(* LS Electric XG5000 project: PID_project *)
(* PLC LSPLC *)
(* module base 0 slot 0: Input/Output Module:XEM-DN/DP32HP (DC 24V Input, Transistor Output, 32 Contacts) *)
(* module base 0 slot 1: Internal Positioning:XBF-PO06E (Open Collector Type, 6 Axis) *)
(* module base 0 slot 2: Input Module:XBE-DC16A/B (DC 24V Input, 16 Contacts / DC12/24V Input, 16 Contacts) *)
(* module base 0 slot 3: Output Module:XBE-RY16A (Relay Output, 16 Contacts (2A, No Varistor/Varistor)) *)
(* module base 0 slot 4: Analog Input Module:XBF-AD04C (A/D Voltage/Current Input Type, 4 Channels, 14bit) *)
(* module base 0 slot 5: Analog Output Module:XBF-DV04C (D/A Voltage Output Type, 4 Channels, 14bit) *)
VAR_GLOBAL
    _04_CH0_DATA AT %UW0.4.2 : WORD; (* Analog Input Module: CH0 Output *)
    _05_CH0_DATA AT %UW0.5.3 : WORD; (* Analog Output Module: CH0 Input *)
    _05_CH0_OUTEN AT %UX0.5.32 : BOOL; (* Analog Output Module: CH0 Output Enable *)
END_VAR

PROGRAM PID_ST (* task: Scan Program *)
(* PID program example in ST *)
VAR RETAIN
    D0_Saved_Value : REAL := 0; (* D value from auto-tune for PID0.  It is a retained variable. *)
    I0_Saved_Value : REAL := 0; (* I value from auto-tune for PID0.  It is a retained variable *)
    P0_Saved_Value : REAL := 1.0; (* P value from auto-tune for PID0.  It is a retained variable *)
    PID0_AutoTune_Completed : BOOL; (* status that auto-tune has been done for PID0.  It is a retained variable. *)
END_VAR
VAR
    Enable_PID0 : BOOL; (* command to enable PID0 *)
    INST_PID0AT : PIDAT; (* instance of auto-tune function block *)
    INST_PID0RUN : PIDRUN; (* instance of PID0 run function block *)
    INST_R_TRIG : R_TRIG;
    PID0_AutoTune_Status : WORD; (* status word of the auto-tune function *)
    PID0_Status : WORD; (* status word of PID0 *)
    Program_Step : USINT := 0; (* program step for PID0 *)
    Rising_Edge_AutoTune : BOOL; (* rising edge of auto-tune command *)
    Run_Auto_Tune : BOOL; (* command to run auto tune *)
END_VAR
VAR_EXTERNAL
    _04_CH0_DATA : WORD; (* AT %UW0.4.2 *) (* Analog Input Module: CH0 Output *)
    _05_CH0_DATA : WORD; (* AT %UW0.5.3 *) (* Analog Output Module: CH0 Input *)
    _05_CH0_OUTEN : BOOL; (* AT %UX0.5.32 *) (* Analog Output Module: CH0 Output Enable *)
END_VAR
(* 
AutomationDirect.com has provided this code for convenience. This sample code is provided "as-is" with no expressed or implied warranty. 
 If the end user includes any of the sample code (in whole or part), it is the user's responsibility to completely modify, integrate, and test any code to ensure it meets all system and 
 safety requirements for the intended application or system.
 *)

//Enable Analog Out CH0 to use it.
_05_CH0_OUTEN := TRUE;

// Clear Analog Out CH0 value if PID0 is disabled.
IF(Enable_PID0 = FALSE) THEN
	_05_CH0_DATA := 0;
END_IF;	

//Moves motor value from analog input ch0 in slot4 to auto-tuning Loop0 current value input device and PID Loop 0 current value input device.
_AT00_PV := _04_CH0_DATA;
_PID00_PV := _04_CH0_DATA;

 INST_R_TRIG(CLK:=Run_Auto_Tune, Q=>Rising_Edge_AutoTune);

CASE Program_Step OF 	
	//Program Step0:  Wait for PID0_Enable to be high.  If auto-tune has been completed, go to PID control in step 50.  If not complete, perform auto-tune in step 10.
	0:
		IF  (Rising_Edge_AutoTune = TRUE) THEN
			Program_Step := 10;
			
		ELSIF (Enable_PID0 = TRUE) AND (PID0_AutoTune_Completed = TRUE) THEN
			Program_Step := 50;
			
		END_IF;	
		
	//Program Step 10: Start Auto-Tune for PID0.  Also, moves output of auto-tuning to CH0 data of analog output module. When Complete go to Step 20.	
	10:	
		_AT00_SV := 2500;  //users set this to a value appropriate for your system
		INST_PID0AT(REQ:=TRUE, BLOCK:=0, LOOP:=0, AT_STAT=>PID0_AutoTune_Status);
		_05_CH0_DATA := _AT00_MV;
		
		IF (_AT00_STATUS = 128) THEN
			PID0_AutoTune_Completed := TRUE;
			Program_Step := 20;
		END_IF;	
	
	//Program Step 20:  Save Auto-tune values to retained variables.  return to step 0 because auto-tune is complete
	20:	
		P0_Saved_Value := _AT00_K_p;
		I0_Saved_Value := _AT00_T_i;
		D0_Saved_Value := _AT00_T_d;
		Program_Step := 0;
		
	//Program Step 50:  Copy saved auto-tune values to PID0 P,I,D values.  move to step 60 to start PID0.	
	50:
		_PID00_K_p := P0_Saved_Value;
		_PID00_T_i := I0_Saved_Value;
		_PID00_T_d := D0_Saved_Value;
		Program_Step := 60;
		
	//Program Step 60: Start the operation of PID Loop0. Copy PID0_MV to analog out CH0 output.  if PID0_Enable is false, go to step 0.	
	60:
		INST_PID0RUN(REQ:=TRUE, BLOCK:=0, LOOP:=0, PID_STAT=>PID0_Status);
		_05_CH0_DATA := _PID00_MV;
		
		IF (Enable_PID0 = FALSE) THEN
			Program_Step := 0;
		
		ELSIF  (Rising_Edge_AutoTune = TRUE) THEN
			Program_Step := 10;		
		END_IF;	
		
END_CASE;
END_PROGRAM

PROGRAM PID_LD (* task: Scan Program *)
(* pid example in ladder *)
VAR RETAIN
    D0_Saved_Value : REAL; (* D value from auto-tune for PID0.  It is a retained variable. *)
    I0_Saved_Value : REAL; (* I value from auto-tune for PID0.  It is a retained variable *)
    P0_Saved_Value : REAL; (* P value from auto-tune for PID0.  It is a retained variable *)
    PID0_AutoTune_Completed : BOOL; (* status that auto-tune has been done for PID0.  It is a retained variable. *)
END_VAR
VAR
    Enable_PID0 : BOOL; (* command to enable PID0 *)
    INST_PID0AT : PIDAT; (* instance of auto-tune function block *)
    INST_PID0RUN : PIDRUN; (* instance of PID0 run function block *)
    PID0_AutoTune_Status : WORD; (* status word of the auto-tune function *)
    PID0_Status : WORD; (* status word of PID0 *)
    Program_Step : USINT := 0; (* program step for PID0 *)
    Run_Auto_Tune : BOOL; (* command to run auto tune *)
END_VAR
VAR_EXTERNAL
    _04_CH0_DATA : WORD; (* AT %UW0.4.2 *) (* Analog Input Module: CH0 Output *)
    _05_CH0_DATA : WORD; (* AT %UW0.5.3 *) (* Analog Output Module: CH0 Input *)
    _05_CH0_OUTEN : BOOL; (* AT %UX0.5.32 *) (* Analog Output Module: CH0 Output Enable *)
END_VAR
VAR
    _e1 : R_TRIG;
    _p2 : BOOL;
    _t3 : BOOL;
    _p4 : BOOL;
    _e5 : R_TRIG;
END_VAR

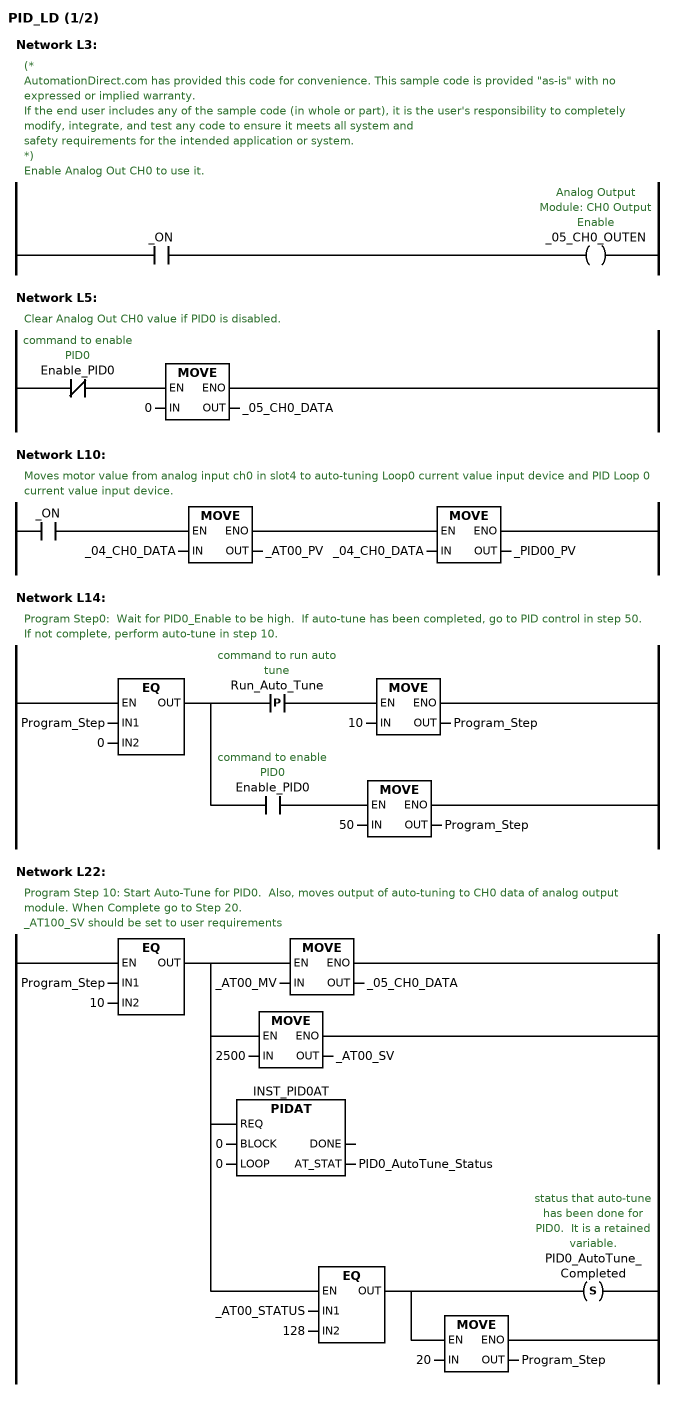
(* ( * / AutomationDirect.com has provided this code for convenience. This sample code is provided "as-is" with no expressed or implied warranty. / If the end user includes any of the sample code (in whole or part), it is the user's responsibility to completely modify, integrate, and test any code to ensure it meets all system and / safety requirements for the intended application or system. / * ) *)
(* Enable Analog Out CH0 to use it. *)
(* Rung L3 *)
_05_CH0_OUTEN := _ON;
(* Clear Analog Out CH0 value if PID0 is disabled. *)
(* Rung L5 *)
IF NOT Enable_PID0 THEN _05_CH0_DATA := 0; END_IF;
(* Moves motor value from analog input ch0 in slot4 to auto-tuning Loop0 current value input device and PID Loop 0 current value input device. *)
(* Rung L10 *)
IF _ON THEN
    _AT00_PV := _04_CH0_DATA;
    _PID00_PV := _04_CH0_DATA;
END_IF;
(* Program Step0:  Wait for PID0_Enable to be high.  If auto-tune has been completed, go to PID control in step 50.  If not complete, perform auto-tune in step 10. *)
(* Rung L14 *)
_e1(CLK := Run_Auto_Tune);
_p2 := Program_Step = 0;
IF (Program_Step = 0) AND _e1.Q THEN Program_Step := 10; END_IF;
IF _p2 AND Enable_PID0 THEN Program_Step := 50; END_IF;
(* Program Step 10: Start Auto-Tune for PID0.  Also, moves output of auto-tuning to CH0 data of analog output module. When Complete go to Step 20. / _AT100_SV should be set to user requirements *)
(* Rung L22 *)
IF Program_Step = 10 THEN
    _05_CH0_DATA := _AT00_MV;
    _AT00_SV := 2500;
END_IF;
INST_PID0AT(REQ := Program_Step = 10, BLOCK := 0, LOOP := 0, AT_STAT => PID0_AutoTune_Status);
IF Program_Step = 10 THEN _t3 := _AT00_STATUS = 128; END_IF;
IF _t3 THEN
    PID0_AutoTune_Completed := TRUE;
    Program_Step := 20;
END_IF;

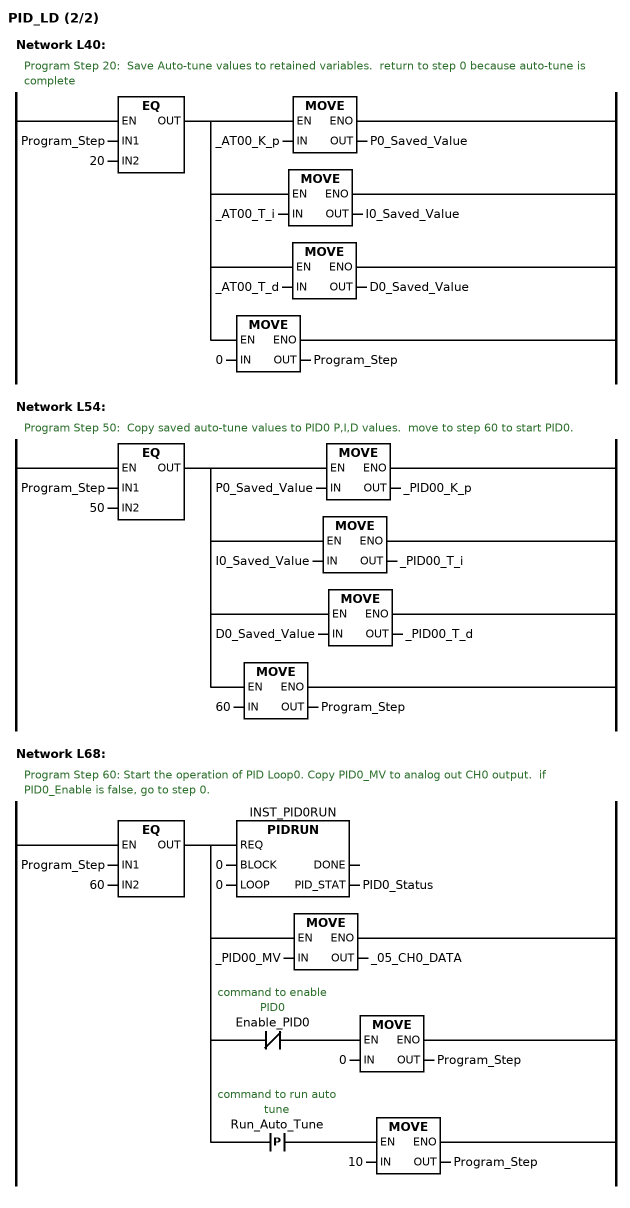
(* Program Step 20:  Save Auto-tune values to retained variables.  return to step 0 because auto-tune is complete *)
(* Rung L40 *)
IF Program_Step = 20 THEN
    P0_Saved_Value := _AT00_K_p;
    I0_Saved_Value := _AT00_T_i;
    D0_Saved_Value := _AT00_T_d;
    Program_Step := 0;
END_IF;
(* Program Step 50:  Copy saved auto-tune values to PID0 P,I,D values.  move to step 60 to start PID0. *)
(* Rung L54 *)
IF Program_Step = 50 THEN
    _PID00_K_p := P0_Saved_Value;
    _PID00_T_i := I0_Saved_Value;
    _PID00_T_d := D0_Saved_Value;
    Program_Step := 60;
END_IF;
(* Program Step 60: Start the operation of PID Loop0. Copy PID0_MV to analog out CH0 output.  if PID0_Enable is false, go to step 0. *)
(* Rung L68 *)
INST_PID0RUN(REQ := Program_Step = 60, BLOCK := 0, LOOP := 0, PID_STAT => PID0_Status);
IF Program_Step = 60 THEN _05_CH0_DATA := _PID00_MV; END_IF;
_p4 := Program_Step = 60;
IF (Program_Step = 60) AND NOT Enable_PID0 THEN Program_Step := 0; END_IF;
_e5(CLK := Run_Auto_Tune);
IF _p4 AND _e5.Q THEN Program_Step := 10; END_IF;
END_PROGRAM